// TIA Portal V18 export
// export: Created 2026-06-21T12:15:02Z, ExportSetting WithDefaults
PlcWatchTable "WT_PLC2_Fake_PLC1_Modbus_Command"
  PlcWatchTableEntry ""DB_Modbus_Holding_Register_DB".CmdSeq"
  PlcWatchTableEntry ""DB_Modbus_Holding_Register_DB".Cmd_Start"
  PlcWatchTableEntry ""DB_Modbus_Holding_Register_DB".Cmd_Stop"
  PlcWatchTableEntry ""DB_Modbus_Holding_Register_DB".Cmd_Reset"
  PlcWatchTableEntry ""DB_Modbus_Holding_Register_DB".Cmd_EStop"
  PlcWatchTableEntry ""DB_Modbus_Holding_Register_DB".Cmd_Load_Recipe"
  PlcWatchTableEntry ""DB_Modbus_Holding_Register_DB".Heartbeat_Client"
  PlcWatchTableEntry ""DB_Modbus_Holding_Register_DB".AckSeq"
  PlcWatchTableEntry ""DB_Modbus_Holding_Register_DB".Done_Branch2"
  PlcWatchTableEntry ""DB_Modbus_Holding_Register_DB".Done_Discharge2"
  PlcWatchTableEntry ""DB_Modbus_Holding_Register_DB".Alarm"
  PlcWatchTableEntry ""DB_Modbus_Holding_Register_DB".State"
